{attribute 'qualified_only'}
VAR_GLOBAL CONSTANT
  MaxDoFs : INT := 7;
  MaxIterations : BYTE := 127; // Maximum iterations when [shrinking an interval](xref:Struckig.Roots#ShrinkInterval)
END_VAR

(* stored: Version 1.1.0.1, ProductVersion 3.1.4024.9
   GVL ParameterList: Id {6cef246a-2041-4266-a931-0bae0d434120}, ParameterList True *)
